INTERFACE I_CommandFeedbackReadWrite EXTENDS I_CommandFeedback, I_CommandBusyState, I_CommandAbortingState

METHOD PUBLIC SetBusy
VAR_INPUT
END_VAR
END_METHOD

END_INTERFACE

(* stored: Version 1.1.0.1, ProductVersion 3.1.4024.12
   Itf I_CommandFeedbackReadWrite: Id {2691a8b1-1544-41ef-976d-1b32800c8e52}
   Method SetBusy: Id {93d3b7cd-e7ce-44b8-a9f8-94592c7cfb5a} *)
